// TIA Portal project "DemoProject" (V17)

(* hardware
DEVICE "PLC_1"  S7-1200 Station
   slot 0: "Rack_0"  S7-1200 Rack  Rack  V1.0
   slot 1: "PLC_1"  CPU 1214C DC/DC/DC  6ES7 214-1AG40-0XB0  V4.5
*)

// ===== PLC "PLC_1"  CPU 1214C DC/DC/DC =====

VAR_GLOBAL   // PLC tag table "IO_Tags"
   "StartBtn" AT %I0.0 : Bool;
   "StopBtn" AT %I0.1 : Bool;
   "MotorRun" AT %Q0.0 : Bool;
   "MotorFault" AT %I0.2 : Bool;
   "AlarmLamp" AT %Q0.1 : Bool;
END_VAR

DATA_BLOCK "DB_Control"   // DB1
{ S7_Optimized_Access := 'TRUE' }
VERSION : 0.1
   VAR
      RunEnable : Bool;   // 运行使能
      FaultAck : Bool;   // 故障确认
      MotorTimer : IEC_TIMER;   // 电机延时定时器
      DelayTime : Time := T#5S;   // 延时时间
   END_VAR
BEGIN
END_DATA_BLOCK

FUNCTION "MotorControl" : Void   // FC1, LAD
{ S7_Optimized_Access := 'TRUE' }
VERSION : 0.1
BEGIN

REGION Network 1
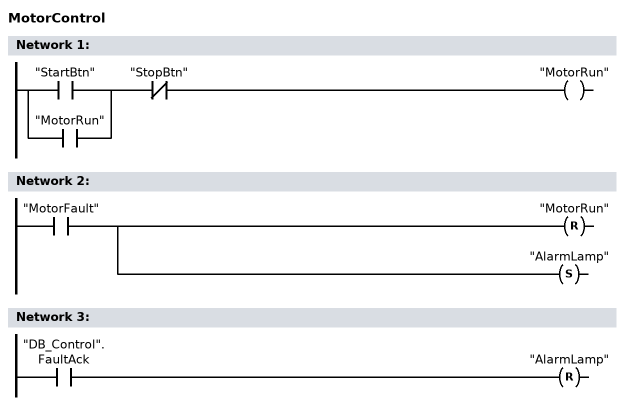
   RUNG wire#powerrail
      Contact( "StartBtn" )
      wire#w1
      I_Contact( "StopBtn" )
      Coil( "MotorRun" )
   END_RUNG
   RUNG wire#powerrail
      Contact( "MotorRun" )
   END_RUNG wire#w1
   // the same network as SCL:
   "MotorRun" := ("StartBtn" OR "MotorRun") AND NOT "StopBtn";
END_REGION

REGION Network 2
   RUNG wire#powerrail
      Contact( "MotorFault" )
      wire#w1
      R_Coil( "MotorRun" )
   END_RUNG
   RUNG wire#w1
      S_Coil( "AlarmLamp" )
   END_RUNG
   // the same network as SCL:
   IF "MotorFault" THEN
       "MotorRun" := FALSE;
       "AlarmLamp" := TRUE;
   END_IF;
END_REGION

REGION Network 3
   RUNG wire#powerrail
      Contact( "DB_Control".FaultAck )
      R_Coil( "AlarmLamp" )
   END_RUNG
   // the same network as SCL:
   IF "DB_Control".FaultAck THEN "AlarmLamp" := FALSE; END_IF;
END_REGION
END_FUNCTION

ORGANIZATION_BLOCK "Main"   // OB1, LAD, ProgramCycle
TITLE = "Main Program Sweep (Cycle)"
{ S7_Optimized_Access := 'TRUE' }
VERSION : 0.1
   VAR_INPUT
      Initial_Call : Bool;   // Initial call of this OB
      Remanence : Bool;   // =True, if remanent data are available
   END_VAR
BEGIN
END_ORGANIZATION_BLOCK